ABB RAPID module: SorterPosition.mod

MODULE SorterPosition
    CONST orient BUFFERPICKUPANGLE := [0.48988,0.48754,0.45322,-0.56295];
    CONST orient SHAKEANGLE := [0.72990,-0.68122,-0.01604,-0.05398];
    CONST orient TABLETANGLE := [0.75194,0.03104,0.65798,-0.02623];

    CONST robtarget PICKUP := [ [-93.5, -560, 215],BUFFERPICKUPANGLE, [0,0,-1,1], [9E9,9E9,9E9,9E9,9E9,9E9] ];
    CONST robtarget DROP := [ [178.2, -355.1, 294.2], BUFFERPICKUPANGLE, [0,0,-1,1], [9E9,9E9,9E9,9E9,9E9,9E9] ];

    CONST robtarget SAFEPOSITION := [ [-57.6, -350, 450], BUFFERPICKUPANGLE, [0,0,-1,1], [9E9,9E9,9E9,9E9,9E9,9E9] ];

     CONST robtarget SORTREST := [ [276.1, -57, 450], TABLETANGLE, [0,0,-1,1], [9E9,9E9,9E9,9E9,9E9,9E9] ];
     CONST robtarget PRESHAKE := [ [209.1,-57, 209.9], SHAKEANGLE, [0,0,-1,1], [9E9,9E9,9E9,9E9,9E9,9E9] ];
     CONST robtarget SHAKEONE := [ [402.6, -57, 209.9], SHAKEANGLE, [0,0,-1,1], [9E9,9E9,9E9,9E9,9E9,9E9] ];
     CONST robtarget SHAKETWO := [ [552.6, -57, 209.9], SHAKEANGLE, [0,0,-1,1], [9E9,9E9,9E9,9E9,9E9,9E9] ];

     CONST robtarget PRETABLETPICKUP := [ [276.1, 120.4, 450],  TABLETANGLE, [0,0,-1,1], [9E9,9E9,9E9,9E9,9E9,9E9] ];
     CONST robtarget TABLETPICKUP := [[404.1, 61.3, 156.8],  TABLETANGLE, [0,0,-1,1], [9E9,9E9,9E9,9E9,9E9,9E9] ];

     CONST robtarget BUFFERSLOT := [ [211.9, -264.2, 310], BUFFERPICKUPANGLE, [0,0,-1,1], [9E9,9E9,9E9,9E9,9E9,9E9] ];
ENDMODULE
